(* CODESYS project Warehouse.project

Project tree, tasks and I/O mapping:
  PLC_AC500_V2 : AC500 PM554-ETH, ABB AG, order no. 1SAP120600R0071, version 2.14.0.0
      settings: PM5xx Type = PM554-ETH; CoDeSys V2.3 Target = 23844; Product version = [2, 2, 0, 5]
    Application
      application App
        global variables GVL
    OBIO : 8DI+6DO, ABB AG, version 2.14.0.0
        unmapped channels: Digital inputs DI0 - DI7, Interrupt DI0 - DI3, State Byte PWM 2, State Byte PWM 3, Unused, Unused, Unused, Unused, Unused, Unused, Unused, Unused, Unused, Unused, Unused, Unused, Unused, Unused, Unused, Actual value 1, Actual value 2, State Byte 1, State Byte 2, Digital outputs DO0 / NO0 - DO5 / NO5, Control Byte PWM 2, PWM 2, frequency / cycle time, PWM 2, duty cycle / duty time, Control Byte PWM 3, Unused, PWM 3, frequency / cycle time, PWM 3, duty cycle / duty time, Unused, Unused, Unused, Unused, Unused, Unused, Unused, Unused, Unused,
          Unused, Unused, Unused, Start value 1, End value 1, Start value 2, End value 2, Control Byte 1, Control Byte 2
    IO_Bus : I/O-Bus, ABB AG, version 2.14.0.0
      DC532 : DC532, ABB AG, order no. 1SAPx40100R0001, version 2.14.0.0
          input  XposRight : BOOL  // Digital inputs I0 - I15.Bytes.Digital inputs I0 - I7.Digital input I0
          input  XposMid : BOOL  // Digital inputs I0 - I15.Bytes.Digital inputs I0 - I7.Digital input I1
          input  XposLeft : BOOL  // Digital inputs I0 - I15.Bytes.Digital inputs I0 - I7.Digital input I2
          input  YposIn : BOOL  // Digital inputs I0 - I15.Bytes.Digital inputs I0 - I7.Digital input I3
          input  YposMid : BOOL  // Digital inputs I0 - I15.Bytes.Digital inputs I0 - I7.Digital input I4
          input  YposOut : BOOL  // Digital inputs I0 - I15.Bytes.Digital inputs I0 - I7.Digital input I5
          input  Zpos3Above : BOOL  // Digital inputs I0 - I15.Bytes.Digital inputs I0 - I7.Digital input I6
          input  Zpos3Below : BOOL  // Digital inputs I0 - I15.Bytes.Digital inputs I0 - I7.Digital input I7
          input  Zpos2Above : BOOL  // Digital inputs I0 - I15.Bytes.Digital inputs I8 - I15.Digital input I8
          input  Zpos2Below : BOOL  // Digital inputs I0 - I15.Bytes.Digital inputs I8 - I15.Digital input I9
          input  Zpos1Above : BOOL  // Digital inputs I0 - I15.Bytes.Digital inputs I8 - I15.Digital input I10
          input  Zpos1Below : BOOL  // Digital inputs I0 - I15.Bytes.Digital inputs I8 - I15.Digital input I11
          input  FeederOccupied : BOOL  // Digital inputs I0 - I15.Bytes.Digital inputs I8 - I15.Digital input I12
          input  Handkey1 : BOOL  // Digital inputs I0 - I15.Bytes.Digital inputs I8 - I15.Digital input I13
          input  Handkey2 : BOOL  // Digital inputs I0 - I15.Bytes.Digital inputs I8 - I15.Digital input I14
          output XRight : BOOL  // Digital outputs C16 - C31.Bytes.Digital outputs C24 - C31.Digital output C24
          output XLeft : BOOL  // Digital outputs C16 - C31.Bytes.Digital outputs C24 - C31.Digital output C25
          output YIn : BOOL  // Digital outputs C16 - C31.Bytes.Digital outputs C24 - C31.Digital output C26
          output YOut : BOOL  // Digital outputs C16 - C31.Bytes.Digital outputs C24 - C31.Digital output C27
          output ZUp : BOOL  // Digital outputs C16 - C31.Bytes.Digital outputs C24 - C31.Digital output C28
          output ZDown : BOOL  // Digital outputs C16 - C31.Bytes.Digital outputs C24 - C31.Digital output C29
          output Led1 : BOOL  // Digital outputs C16 - C31.Bytes.Digital outputs C24 - C31.Digital output C30
          output Led2 : BOOL  // Digital outputs C16 - C31.Bytes.Digital outputs C24 - C31.Digital output C31
          unmapped channels: Digital inputs I0 - I15, Digital inputs C16 - C31, Digital outputs C16 - C31, Actual value 1, Actual value 2, State Byte 1, State Byte 2, Start value 1, End value 1, Start value 2, End value 2, Control Byte 1, Control Byte 2, Digital inputs I0 - I15, Digital inputs C16 - C31, Digital outputs C16 - C31, Digital inputs I0 - I15, Digital inputs C16 - C31, Digital outputs C16 - C31
    Interfaces : Interfaces, ABB AG, version 2.14.0.0
      COM1_Online_Access : COM1 - Online Access, ABB AG, version 2.14.0.0
      COM2_None : COM2 - None, ABB AG, version 2.14.0.0
      Ethernet : Onboard Ethernet, ABB AG, version 2.14.0.0
        ETH1 : ETH1, ABB AG, version 2.14.0.0
        Protocols : Protocols, ABB AG, version 2.14.0.0
  libraries: VisuSymbols, 4.5.0.0 (System)
  visualisation Visualization
  text list GlobalTextList
*)

// PLC_AC500_V2/Application/App/GVL
VAR_GLOBAL
	 inventory:ARRAY[0..3,0..3] OF INT;
	x_sensors: ARRAY[1..3] OF BOOL;
	inp:BOOL:=FALSE;
	pos:INT:=0;
	(*z_sensors_above:ARRAY[Zpose1Above, Zpose2Above, Zpose3Above] OF BOOL;
	z_sensors_below:ARRAY[Zpose1Below, Zpose2Below, Zpose3Below] OF BOOL;*)
	led1ABB:BOOL:=FALSE;
END_VAR

// /Visualization
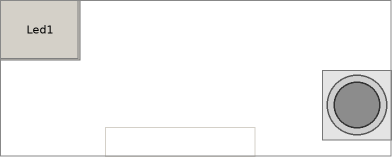
VISUALIZATION Visualization  // 392x157
    PushSwitch (322,70 70x70), behaviour: TOGGLE, style: Switch-PushSwitch-Gray
    Button (0,0 80x60), "Led1"
        toggle led1ABB
    Textfield (105,127 150x30)
END_VISUALIZATION
